// TIA Portal project "FactoryIO_Template_S7-1200_V15_V15.1" (V15.1)
// Vorlageprojekt für das Buch mit Zielsystem S7-1200

(* hardware
DEVICE "S7-1200-Station_1"  S7-1200 Station
   slot 0: "Baugruppenträger_0"  Rack  V1.0
   slot 1: "PLC_1"  CPU 1211C DC/DC/DC  6ES7 211-1AE40-0XB0  V4.1
DEVICE "HMI_1"  KTP900 Basic PN
   slot 0: "HMI_1"  KTP900 Basic PN  6AV2 123-2JB03-0AX0  15.1.0.0
   slot 1: "HMI_RT_1"  KTP900 Basic PN  6AV2 123-2JB03-0AX0  15.1.0.0
   slot 5: "HMI_1.IE_CP_1"  PROFINET Interface  15.0.1.0
      slot 1: "PROFINET Interface_1"  PROFINET Interface
         slot 1: "Port_1"  Port
*)

// ===== PLC "PLC_1"  CPU 1211C DC/DC/DC =====

VAR_GLOBAL   // PLC tag table "Standard-Variablentabelle"
   "Moving X" AT %I0.0 : Bool;
   "Moving Z" AT %I0.1 : Bool;
   "Item detected" AT %I0.2 : Bool;
   "Lid at place" AT %I0.3 : Bool;
   "Lid clamped" AT %I0.4 : Bool;
   "Pos. at limit (lids)" AT %I0.5 : Bool;
   "Base at place" AT %I0.6 : Bool;
   "Base clamped" AT %I0.7 : Bool;
   "Pos. at limit (bases)" AT %I1.0 : Bool;
   "Part leaving" AT %I1.1 : Bool;
   "Start" AT %I1.2 : Bool;
   "Reset" AT %I1.3 : Bool;
   "Stop" AT %I1.4 : Bool;
   "Emergency stop" AT %I1.5 : Bool;
   "Auto" AT %I1.6 : Bool;
   "Running" AT %I1.7 : Bool;
   "Move X" AT %Q0.0 : Bool;
   "Move Z" AT %Q0.1 : Bool;
   "Grab" AT %Q0.2 : Bool;
   "Lids conveyor" AT %Q0.3 : Bool;
   "Clamp lid" AT %Q0.4 : Bool;
   "Pos. raise (lids)" AT %Q0.5 : Bool;
   "Bases conveyor" AT %Q0.6 : Bool;
   "Clamp base" AT %Q0.7 : Bool;
   "Pos. raise (bases)" AT %Q1.0 : Bool;
   "Start light" AT %Q1.1 : Bool;
   "Reset light" AT %Q1.2 : Bool;
   "Stop light" AT %Q1.3 : Bool;
   "Counter" AT %QD30 : DInt;
   "Tag_1" AT %M0.0 : Bool;
   "Tag_2" AT %M0.1 : Bool;
   "Tag_3" AT %M0.2 : Bool;
   "Tag_4" AT %M0.3 : Bool;
   "Tag_5" AT %M0.4 : Bool;
   "Tag_6" AT %M0.5 : Bool;
   "Lid alined" AT %M0.6 : Bool;
   "Tag_7" AT %M0.7 : Bool;
   "Tag_8" AT %M1.0 : Bool;
   "Base alined" AT %M1.1 : Bool;
   "Tag_9" AT %M1.2 : Bool;
   "Move Z bit" AT %M1.3 : Bool;
   "Tag_10" AT %M1.4 : Bool;
   "Tag_11" AT %M1.5 : Bool;
   "Tag_12" AT %M1.6 : Bool;
   "Tag_13" AT %M1.7 : Bool;
   "Tag_14" AT %M2.0 : Bool;
   "Move Z bit 2" AT %M2.1 : Bool;
   "Tag_15" AT %M2.2 : Bool;
   "temp" AT %M2.3 : Bool;
   "Tag_16" AT %M2.4 : Bool;
   "temp_2" AT %M2.5 : Bool;
   "Tag_17" AT %M2.6 : Bool;
END_VAR

DATA_BLOCK "Auxiliare"   // DB1
{ S7_Optimized_Access := 'TRUE' }
VERSION : 0.1
   VAR
      nr_cutii_cerut : USInt;
      nr_cutii_curent : USInt;
      comanda_Start : Bool;
      re1 : Bool;
   END_VAR
BEGIN
END_DATA_BLOCK

// folder: System blocks/Program resources

DATA_BLOCK "timer_grab"   // DB2
{ S7_Optimized_Access := 'TRUE' }
AUTHOR : Simatic
FAMILY : IEC
NAME : IEC_TMR
VERSION : 1.0
// stored: InstanceOfName IEC_TIMER
"IEC_TIMER"
BEGIN
END_DATA_BLOCK

DATA_BLOCK "timer_clamps"   // DB3
{ S7_Optimized_Access := 'TRUE' }
AUTHOR : Simatic
FAMILY : IEC
NAME : IEC_TMR
VERSION : 1.0
// stored: InstanceOfName IEC_TIMER
"IEC_TIMER"
BEGIN
END_DATA_BLOCK

DATA_BLOCK "timer_grab_2"   // DB4
{ S7_Optimized_Access := 'TRUE' }
AUTHOR : Simatic
FAMILY : IEC
NAME : IEC_TMR
VERSION : 1.0
// stored: InstanceOfName IEC_TIMER
"IEC_TIMER"
BEGIN
END_DATA_BLOCK

DATA_BLOCK "timer_ridicare_porti"   // DB5
{ S7_Optimized_Access := 'TRUE' }
AUTHOR : Simatic
FAMILY : IEC
NAME : IEC_TMR
VERSION : 1.0
// stored: InstanceOfName IEC_TIMER
"IEC_TIMER"
BEGIN
END_DATA_BLOCK

// folder: (top level)

FUNCTION "clamp" : Void   // FC1, LAD
{ S7_Optimized_Access := 'TRUE' }
VERSION : 0.1
BEGIN

REGION Network 1: clamp pentru lid
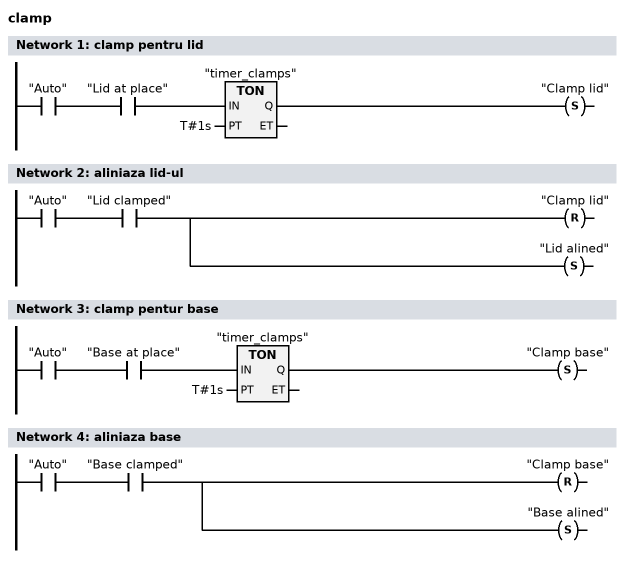
   "timer_clamps".TON(IN := "Auto" AND "Lid at place", PT := T#1s);
   IF "timer_clamps".Q THEN "Clamp lid" := TRUE; END_IF;
END_REGION

REGION Network 2: aliniaza lid-ul
   RUNG wire#powerrail
      Contact( "Auto" )
      Contact( "Lid clamped" )
      wire#w1
      R_Coil( "Clamp lid" )
   END_RUNG
   RUNG wire#w1
      S_Coil( "Lid alined" )
   END_RUNG
   // the same network as SCL:
   IF "Auto" AND "Lid clamped" THEN
       "Clamp lid" := FALSE;
       "Lid alined" := TRUE;
   END_IF;
END_REGION

REGION Network 3: clamp pentur base
   "timer_clamps".TON(IN := "Auto" AND "Base at place", PT := T#1s);
   IF "timer_clamps".Q THEN "Clamp base" := TRUE; END_IF;
END_REGION

REGION Network 4: aliniaza base
   RUNG wire#powerrail
      Contact( "Auto" )
      Contact( "Base clamped" )
      wire#w1
      R_Coil( "Clamp base" )
   END_RUNG
   RUNG wire#w1
      S_Coil( "Base alined" )
   END_RUNG
   // the same network as SCL:
   IF "Auto" AND "Base clamped" THEN
       "Clamp base" := FALSE;
       "Base alined" := TRUE;
   END_IF;
END_REGION
END_FUNCTION

FUNCTION "pick-place" : Void   // FC2, LAD
{ S7_Optimized_Access := 'TRUE' }
VERSION : 0.1
BEGIN

REGION Network 1: muta pe z ca sa ia lid ul
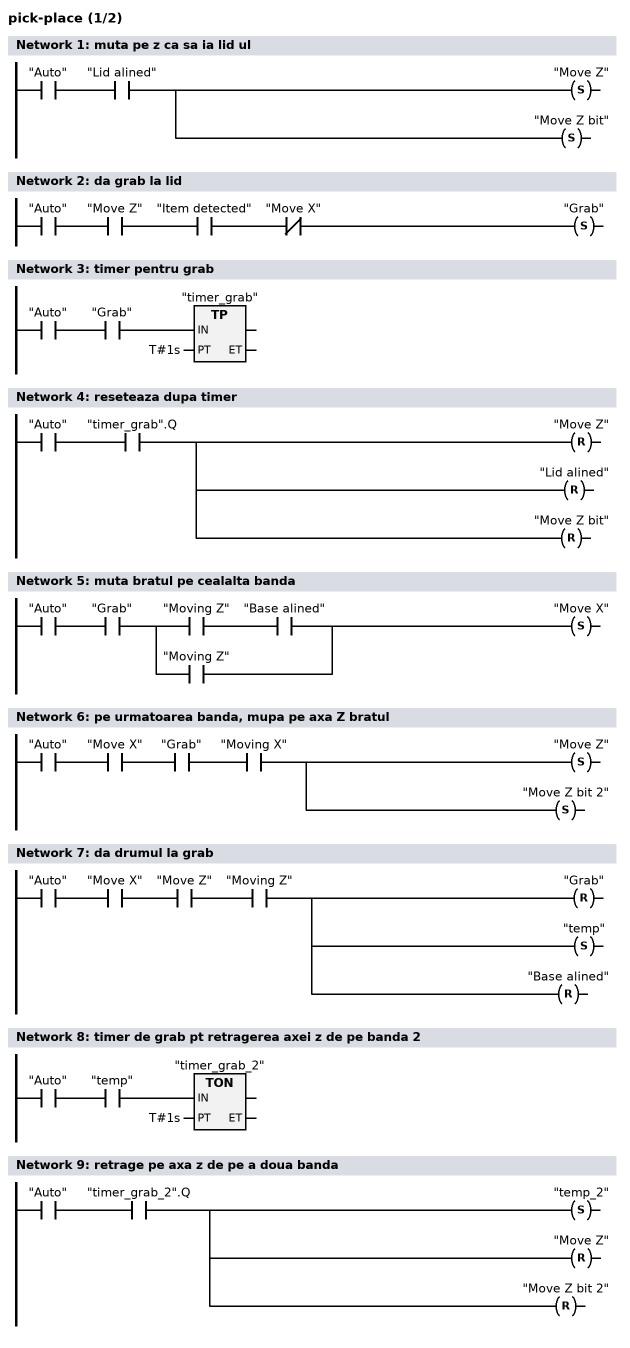
   RUNG wire#powerrail
      Contact( "Auto" )
      Contact( "Lid alined" )
      wire#w1
      S_Coil( "Move Z" )
   END_RUNG
   RUNG wire#w1
      S_Coil( "Move Z bit" )
   END_RUNG
   // the same network as SCL:
   IF "Auto" AND "Lid alined" THEN
       "Move Z" := TRUE;
       "Move Z bit" := TRUE;
   END_IF;
END_REGION

REGION Network 2: da grab la lid
   RUNG wire#powerrail
      Contact( "Auto" )
      Contact( "Move Z" )
      Contact( "Item detected" )
      I_Contact( "Move X" )
      S_Coil( "Grab" )
   END_RUNG
   // the same network as SCL:
   IF "Auto" AND "Move Z" AND "Item detected" AND NOT "Move X" THEN "Grab" := TRUE; END_IF;
END_REGION

REGION Network 3: timer pentru grab
   "timer_grab".TP(IN := "Auto" AND "Grab", PT := T#1s);
END_REGION

REGION Network 4: reseteaza dupa timer
   RUNG wire#powerrail
      Contact( "Auto" )
      Contact( "timer_grab".Q )
      wire#w1
      R_Coil( "Move Z" )
   END_RUNG
   RUNG wire#w1
      R_Coil( "Lid alined" )
   END_RUNG
   RUNG wire#w1
      R_Coil( "Move Z bit" )
   END_RUNG
   // the same network as SCL:
   IF "Auto" AND "timer_grab".Q THEN
       "Move Z" := FALSE;
       "Lid alined" := FALSE;
       "Move Z bit" := FALSE;
   END_IF;
END_REGION

REGION Network 5: muta bratul pe cealalta banda
   RUNG wire#powerrail
      Contact( "Auto" )
      Contact( "Grab" )
      wire#w1
      Contact( "Moving Z" )
      Contact( "Base alined" )
      wire#w2
      S_Coil( "Move X" )
   END_RUNG
   RUNG wire#w1
      Contact( "Moving Z" )
   END_RUNG wire#w2
   // the same network as SCL:
   IF "Auto" AND "Grab" AND (("Moving Z" AND "Base alined") OR "Moving Z") THEN "Move X" := TRUE; END_IF;
END_REGION

REGION Network 6: pe urmatoarea banda, mupa pe axa Z bratul
   RUNG wire#powerrail
      Contact( "Auto" )
      Contact( "Move X" )
      Contact( "Grab" )
      Contact( "Moving X" )
      wire#w1
      S_Coil( "Move Z" )
   END_RUNG
   RUNG wire#w1
      S_Coil( "Move Z bit 2" )
   END_RUNG
   // the same network as SCL:
   IF "Auto" AND "Move X" AND "Grab" AND "Moving X" THEN
       "Move Z" := TRUE;
       "Move Z bit 2" := TRUE;
   END_IF;
END_REGION

REGION Network 7: da drumul la grab
   RUNG wire#powerrail
      Contact( "Auto" )
      Contact( "Move X" )
      Contact( "Move Z" )
      Contact( "Moving Z" )
      wire#w1
      R_Coil( "Grab" )
   END_RUNG
   RUNG wire#w1
      S_Coil( "temp" )
   END_RUNG
   RUNG wire#w1
      R_Coil( "Base alined" )
   END_RUNG
   // the same network as SCL:
   IF "Auto" AND "Move X" AND "Move Z" AND "Moving Z" THEN
       "Grab" := FALSE;
       "temp" := TRUE;
       "Base alined" := FALSE;
   END_IF;
END_REGION

REGION Network 8: timer de grab pt retragerea axei z de pe banda 2
   "timer_grab_2".TON(IN := "Auto" AND "temp", PT := T#1s);
END_REGION

REGION Network 9: retrage pe axa z de pe a doua banda
   RUNG wire#powerrail
      Contact( "Auto" )
      Contact( "timer_grab_2".Q )
      wire#w1
      S_Coil( "temp_2" )
   END_RUNG
   RUNG wire#w1
      R_Coil( "Move Z" )
   END_RUNG
   RUNG wire#w1
      R_Coil( "Move Z bit 2" )
   END_RUNG
   // the same network as SCL:
   IF "Auto" AND "timer_grab_2".Q THEN
       "temp_2" := TRUE;
       "Move Z" := FALSE;
       "Move Z bit 2" := FALSE;
   END_IF;
END_REGION

REGION Network 10: timer pentru ridicarea la porti
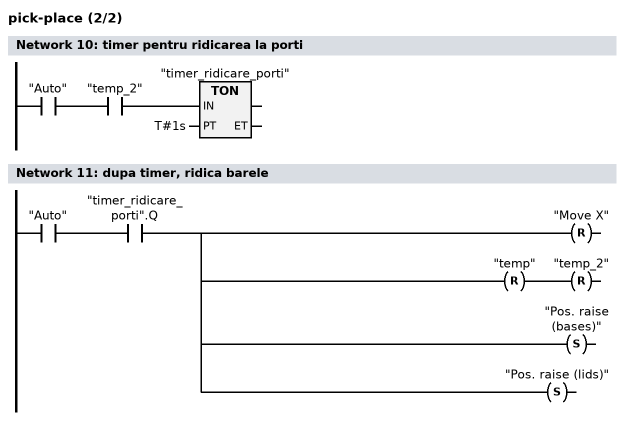
   "timer_ridicare_porti".TON(IN := "Auto" AND "temp_2", PT := T#1s);
END_REGION

REGION Network 11: dupa timer, ridica barele
   RUNG wire#powerrail
      Contact( "Auto" )
      Contact( "timer_ridicare_porti".Q )
      wire#w1
      R_Coil( "Move X" )
   END_RUNG
   RUNG wire#w1
      R_Coil( "temp" )
      R_Coil( "temp_2" )
   END_RUNG
   RUNG wire#w1
      S_Coil( "Pos. raise (bases)" )
   END_RUNG
   RUNG wire#w1
      S_Coil( "Pos. raise (lids)" )
   END_RUNG
   // the same network as SCL:
   IF "Auto" AND "timer_ridicare_porti".Q THEN
       "Move X" := FALSE;
       "temp" := FALSE;
       "temp_2" := FALSE;
       "Pos. raise (bases)" := TRUE;
       "Pos. raise (lids)" := TRUE;
   END_IF;
END_REGION
END_FUNCTION

FUNCTION "belt" : Void   // FC3, LAD
{ S7_Optimized_Access := 'TRUE' }
VERSION : 0.1
BEGIN

REGION Network 1: porneste pe auto benzile
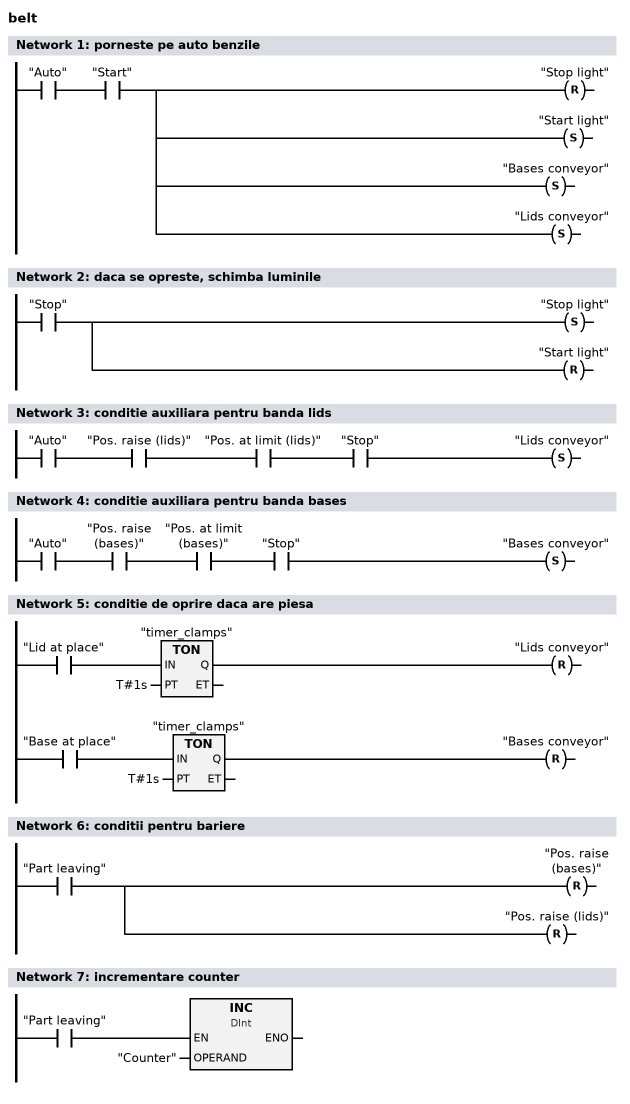
   RUNG wire#powerrail
      Contact( "Auto" )
      Contact( "Start" )
      wire#w1
      R_Coil( "Stop light" )
   END_RUNG
   RUNG wire#w1
      S_Coil( "Start light" )
   END_RUNG
   RUNG wire#w1
      S_Coil( "Bases conveyor" )
   END_RUNG
   RUNG wire#w1
      S_Coil( "Lids conveyor" )
   END_RUNG
   // the same network as SCL:
   IF "Auto" AND "Start" THEN
       "Stop light" := FALSE;
       "Start light" := TRUE;
       "Bases conveyor" := TRUE;
       "Lids conveyor" := TRUE;
   END_IF;
END_REGION

REGION Network 2: daca se opreste, schimba luminile
   RUNG wire#powerrail
      Contact( "Stop" )
      wire#w1
      S_Coil( "Stop light" )
   END_RUNG
   RUNG wire#w1
      R_Coil( "Start light" )
   END_RUNG
   // the same network as SCL:
   IF "Stop" THEN
       "Stop light" := TRUE;
       "Start light" := FALSE;
   END_IF;
END_REGION

REGION Network 3: conditie auxiliara pentru banda lids
   RUNG wire#powerrail
      Contact( "Auto" )
      Contact( "Pos. raise (lids)" )
      Contact( "Pos. at limit (lids)" )
      Contact( "Stop" )
      S_Coil( "Lids conveyor" )
   END_RUNG
   // the same network as SCL:
   IF "Auto" AND "Pos. raise (lids)" AND "Pos. at limit (lids)" AND "Stop" THEN
       "Lids conveyor" := TRUE;
   END_IF;
END_REGION

REGION Network 4: conditie auxiliara pentru banda bases
   RUNG wire#powerrail
      Contact( "Auto" )
      Contact( "Pos. raise (bases)" )
      Contact( "Pos. at limit (bases)" )
      Contact( "Stop" )
      S_Coil( "Bases conveyor" )
   END_RUNG
   // the same network as SCL:
   IF "Auto" AND "Pos. raise (bases)" AND "Pos. at limit (bases)" AND "Stop" THEN
       "Bases conveyor" := TRUE;
   END_IF;
END_REGION

REGION Network 5: conditie de oprire daca are piesa
   "timer_clamps".TON(IN := "Lid at place", PT := T#1s);
   IF "timer_clamps".Q THEN "Lids conveyor" := FALSE; END_IF;
   "timer_clamps".TON(IN := "Base at place", PT := T#1s);
   IF "timer_clamps".Q THEN "Bases conveyor" := FALSE; END_IF;
END_REGION

REGION Network 6: conditii pentru bariere
   RUNG wire#powerrail
      Contact( "Part leaving" )
      wire#w1
      R_Coil( "Pos. raise (bases)" )
   END_RUNG
   RUNG wire#w1
      R_Coil( "Pos. raise (lids)" )
   END_RUNG
   // the same network as SCL:
   IF "Part leaving" THEN
       "Pos. raise (bases)" := FALSE;
       "Pos. raise (lids)" := FALSE;
   END_IF;
END_REGION

REGION Network 7: incrementare counter
   RUNG wire#powerrail
      Contact( "Part leaving" )
      { S7_Templates := "DestType := DInt" } Inc( "Counter" )
   END_RUNG
   // the same network as SCL:
   IF "Part leaving" THEN "Counter" := "Counter" + 1; END_IF;
END_REGION
END_FUNCTION

FUNCTION "MHJ-PLC-Lab-Function-S71200" : Void   // FC9000, SCL
{ S7_Optimized_Access := 'TRUE' }
VERSION : 0.1
   VAR_TEMP
      rdTimeReturn : Int;
      outputTime : DTL;
      SyncVal : Byte;
      forVal : Int;
      forVal_2 : Int;
      Value : Byte;
   END_VAR
   VAR CONSTANT
      CompVal : Byte := 16#34;
      Value_01 : Byte := 16#11;
      Value_01_DW : DWord := 16#A165_D992;
      Value_02_DW : DWord := 16#58BE_4401;
   END_VAR
BEGIN

   #Value:=PEEK(area := 16#82,
        dbNumber := 0,
        byteOffset := 511);
   #Value := #Value + 1;

   POKE(area := 16#82,
        dbNumber := 0,
        byteOffset := 511,
        value := #Value);

   POKE(area:=16#81,
        dbNumber:=0,
        byteOffset:=1016,
        value:=#Value_01_DW);
   POKE(area := 16#81,
        dbNumber := 0,
        byteOffset := 1020,
        value := #Value_02_DW);

   POKE(area := 16#81,
        dbNumber := 0,
        byteOffset := 511,
        value := B#16#00);

   FOR #forVal := 0 TO 120 DO
       FOR #forVal_2:=0 TO 10 DO
           #rdTimeReturn:=RD_SYS_T(#outputTime);
           #rdTimeReturn := WR_SYS_T(#outputTime);
           #rdTimeReturn := RD_SYS_T(#outputTime);
           #rdTimeReturn := WR_SYS_T(#outputTime);
       END_FOR;
       #SyncVal:= PEEK(area := 16#81,
                      dbNumber := 0,
                      byteOffset := 511);
       IF #SyncVal = #CompVal THEN
          GOTO M_1;
       END_IF;
   END_FOR;
   RETURN;

   M_1:
   POKE(area := 16#81,
        dbNumber := 0,
        byteOffset := 511,
        value := B#16#0);
END_FUNCTION

ORGANIZATION_BLOCK "Main"   // OB1, LAD, ProgramCycle
TITLE = "Main Program Sweep (Cycle)"
{ S7_Optimized_Access := 'TRUE' }
VERSION : 0.1
   VAR_INPUT
      Initial_Call : Bool;   // Initial call of this OB
      Remanence : Bool;   // =True, if remanent data are available
   END_VAR
BEGIN

REGION Network 1: Konnektierungsbaustein für PLC-Lab
   // Im Netzwerk 1 wird der Konnektierungsbaustein für PLC-Lab aufgerufen.
   // Dieser Aufruf darf nicht entfernt werden!
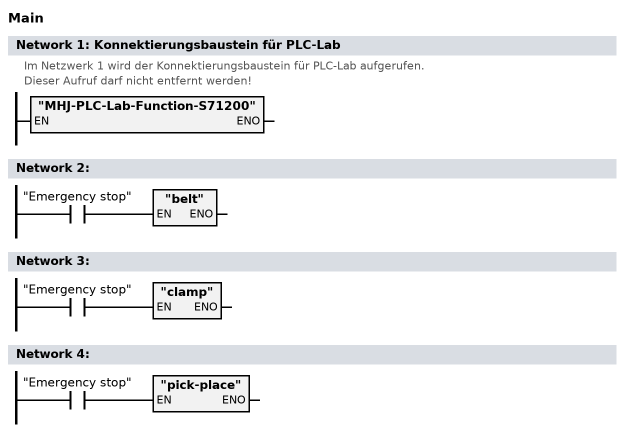
   RUNG wire#powerrail
      "MHJ-PLC-Lab-Function-S71200"()
   END_RUNG
   // the same network as SCL:
   "MHJ-PLC-Lab-Function-S71200"();
END_REGION

REGION Network 2
   RUNG wire#powerrail
      Contact( "Emergency stop" )
      "belt"()
   END_RUNG
   // the same network as SCL:
   IF "Emergency stop" THEN "belt"(); END_IF;
END_REGION

REGION Network 3
   RUNG wire#powerrail
      Contact( "Emergency stop" )
      "clamp"()
   END_RUNG
   // the same network as SCL:
   IF "Emergency stop" THEN "clamp"(); END_IF;
END_REGION

REGION Network 4
   RUNG wire#powerrail
      Contact( "Emergency stop" )
      "pick-place"()
   END_RUNG
   // the same network as SCL:
   IF "Emergency stop" THEN "pick-place"(); END_IF;
END_REGION
END_ORGANIZATION_BLOCK

(* ===== HMI "HMI_RT_1" =====
system functions are stored by id; their names below are inferred from use
connection "HMI_Connection_1": ETHERNET, SMART_S7_1200_OMS

HMI tags "Default tag table"
   "Fill" : Bool = PLC Item_ready AT %I0.0, 1 s
   "Discharge" : Bool = PLC At_entry AT %I0.1, 1 s
   "running" : Bool = PLC Running AT %I1.7, 1 s
   "Auxiliare_nr_cutii_cerut" : USInt = PLC Auxiliare.nr_cutii_cerut, 1 s
   "Auxiliare_comanda_Start" : Bool = PLC Auxiliare.comanda_Start, 1 s
   "Auxiliare_nr_cutii_curent" : USInt = PLC Auxiliare.nr_cutii_curent, 1 s

Template "Template_1" 800x480
   Button "Exit" at 722,440 size 55x39; TextOff 'Exit'; PictureOff "ExitRuntime_KTP900_Basic_PN_TR"; PictureOn "ExitRuntime_KTP900_Basic_PN_TR"
      on Release: StopRuntime(0)
   Button "Template_Button" at 622,440 size 55x39; TextOff 'Text'
   Button "Template_Button_1" at 522,440 size 55x39; TextOff 'Text'
   Button "Template_Button_2" at 422,440 size 55x39; TextOff 'Text'
   Button "Template_Button_3" at 322,440 size 55x39; TextOff 'Text'
   Button "Template_Button_4" at 222,440 size 55x39; TextOff 'Text'
   Button "Template_Button_5" at 122,440 size 55x39; TextOff 'Text'
   Button "Start screen" at 22,440 size 55x39; TextOff 'Start screen'; PictureOff "NavigateHome_KTP900_Basic_PN_TR"; PictureOn "NavigateHome_KTP900_Basic_PN_TR"
      on Release: ActivateScreen("Main", 0)

screen "Main" 800x480, template "Template_1"
   IOField "I/O field_1" at 349,112 size 102x43; FormatPattern 999
      ProcessValue <- "Auxiliare_nr_cutii_cerut"
   TextField "Text field_1" at 369,83 size 62x20; Text 'Nr. cerut'
   Button "Button_1" at 349,176 size 102x38; TextOff 'Pornire'
      on Click: SetBit("Auxiliare_comanda_Start")
   Circle "Circle_1" at 372,230 size 56x56
      Appearance <- "running"
   IOField "I/O field_2" at 352,328 size 96x32; FormatPattern 999
      ProcessValue <- "Auxiliare_nr_cutii_curent"
   TextField "Text field_2" at 366,299 size 70x20; Text 'Nr. curent'
*)